// TIA Portal V19 export
ORGANIZATION_BLOCK "Pull or plug of modules"   // OB83, STL, PullOrPlugOfModules
{ S7_Optimized_Access := 'FALSE' }
   VAR_TEMP
      EV_CLASS : Byte;   // 16#38:Event class 3 - module inserted, 16#39: Event class 3 - module removed
      FLT_ID : Byte;   // Fault identifier
      PRIORITY : Byte;   // Priority of OB Execution
      OB_NUMBR : Byte;   // OB number
      RESERVED_1 : Byte;   // Reserved for system
      MDL_ID : Byte;   // 16#54:input, 16#55:output, 16#0:not available
      MDL_ADDR : Word;   // Hardware identifier
      RACK_NUM : Int;   // Rack number
      MDL_TYPE : Word;   // Module type
      DATE_TIME : Date_And_Time;   // Date and time OB started
   END_VAR
BEGIN
END_ORGANIZATION_BLOCK
